FUNCTION_BLOCK SimpleLiftController
  (* Standard: 61499-2 *)
  (* Version 0.1, 2014-00-16, Canto-Air, CANTO-AIR-PC *)
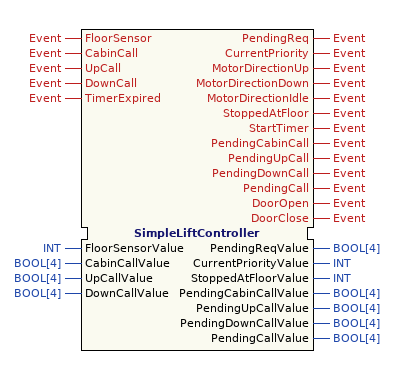
  EVENT_INPUT
    FloorSensor;
    CabinCall;
    UpCall;
    DownCall;
    TimerExpired;
  END_EVENT
  EVENT_OUTPUT
    PendingReq;
    CurrentPriority;
    MotorDirectionUp;
    MotorDirectionDown;
    MotorDirectionIdle;
    StoppedAtFloor;
    StartTimer;
    PendingCabinCall;
    PendingUpCall;
    PendingDownCall;
    PendingCall;
    DoorOpen;
    DoorClose;
  END_EVENT
  VAR_INPUT
    FloorSensorValue : INT;
    CabinCallValue : ARRAY [0..3] OF BOOL;
    UpCallValue : ARRAY [0..3] OF BOOL;
    DownCallValue : ARRAY [0..3] OF BOOL;
  END_VAR
  VAR_OUTPUT
    PendingReqValue : ARRAY [0..3] OF BOOL;
    CurrentPriorityValue : INT;
    StoppedAtFloorValue : INT;
    PendingCabinCallValue : ARRAY [0..3] OF BOOL;
    PendingUpCallValue : ARRAY [0..3] OF BOOL;
    PendingDownCallValue : ARRAY [0..3] OF BOOL;
    PendingCallValue : ARRAY [0..3] OF BOOL;
  END_VAR
  FBS
    UnitControl : UnitControl;
    RequestResolver : RequestResolver;
  END_FBS
  EVENT_CONNECTIONS
    FloorSensor TO UnitControl.FloorSensor;
    FloorSensor TO RequestResolver.FloorSensor;
    CabinCall TO RequestResolver.CabinCall;
    UpCall TO RequestResolver.UpCall;
    DownCall TO RequestResolver.DownCall;
    TimerExpired TO UnitControl.TimerExpired;
    RequestResolver.PendingReq TO PendingReq;
    RequestResolver.CurrentPriority TO CurrentPriority;
    UnitControl.MotorDirectionUp TO MotorDirectionUp;
    UnitControl.MotorDirectionDown TO MotorDirectionDown;
    UnitControl.MotorDirectionIdle TO MotorDirectionIdle;
    UnitControl.StoppedAtFloor TO StoppedAtFloor;
    UnitControl.StartTimer TO StartTimer;
    RequestResolver.PendingCabinCall TO PendingCabinCall;
    RequestResolver.PendingUpCall TO PendingUpCall;
    RequestResolver.PendingDownCall TO PendingDownCall;
    RequestResolver.PendingCall TO PendingCall;
    UnitControl.DoorOpen TO DoorOpen;
    UnitControl.DoorClose TO DoorClose;
    UnitControl.MotorDirectionUp TO RequestResolver.MotorDirectionUp;
    UnitControl.MotorDirectionDown TO RequestResolver.MotorDirectionDown;
    UnitControl.MotorDirectionIdle TO RequestResolver.MotorDirectionIdle;
    UnitControl.StoppedAtFloor TO RequestResolver.StoppedAtFloor;
    RequestResolver.request TO UnitControl.Request;
  END_CONNECTIONS
  DATA_CONNECTIONS
    FloorSensorValue TO UnitControl.FloorSensorValue;
    FloorSensorValue TO RequestResolver.FloorSensorValue;
    CabinCallValue TO RequestResolver.CabinCallValue;
    UpCallValue TO RequestResolver.UpCallValue;
    DownCallValue TO RequestResolver.DownCallValue;
    RequestResolver.PendingReqValue TO PendingReqValue;
    RequestResolver.CurrentPriorityValue TO CurrentPriorityValue;
    UnitControl.StoppedAtFloorValue TO StoppedAtFloorValue;
    RequestResolver.PendingCabinCallValue TO PendingCabinCallValue;
    RequestResolver.PendingUpCallValue TO PendingUpCallValue;
    RequestResolver.PendingDownCallValue TO PendingDownCallValue;
    RequestResolver.PendingCallValue TO PendingCallValue;
    UnitControl.StoppedAtFloorValue TO RequestResolver.StoppedAtFloorValue;
    RequestResolver.requestValue TO UnitControl.RequestValue;
  END_CONNECTIONS
END_FUNCTION_BLOCK
